FUNCTION alg_a_transfer2pickpos : BOOL
VAR_INPUT
	state: STATE;
END_VAR

alg_a_transfer2pickpos := state.dvar_M_vacuum_a_transfer2pickpos;

END_FUNCTION

(* stored: Version 1.1.0.1, ProductVersion 3.1.4022.18
   POU alg_a_transfer2pickpos: Id {e0940764-00a6-4f9d-9f26-ac3f313d6991}, SpecialFunc None *)
